Fanuc KAREL source: kb00030.KL

PROGRAM KB00030
%STACKSIZE=65535
%PRIORITY=65535
%NOLOCKGROUP
VAR
P1 : INTEGER
P2 : INTEGER
P3 : STRING[80]
P4 : INTEGER
BEGIN
P1=1
P2=1
P3='A'
P4=1
CNC_DYN_DISP(P1,P2,P3,P4)
END KB00030
